Staubli VAL3: MoveJoint.pgx

program MoveJoint(num x_nJ1, num x_nJ2, num x_nJ3, num x_nJ4, num x_nJ5, num x_nJ6)
  local joint l_jJoint
begin
  l_jJoint.j1 = x_nJ1
  l_jJoint.j2 = x_nJ2
  l_jJoint.j3 = x_nJ3
  l_jJoint.j4 = x_nJ4
  l_jJoint.j5 = x_nJ5
  l_jJoint.j6 = x_nJ6
  movej(l_jJoint, tCurrentTool, mCurrentSpeed)
end
